  00:  IF ( _execute_R.Q )  
       THEN
         // Check function is supported and parameter are valid ?
         IF (( CheckFunctionSupported( AxesGroup := AxesGroup )) AND
             ( CheckParameterValid   ( AxesGroup := AxesGroup )))      
         THEN
           // set busy flag
           Busy := TRUE;
           // Reset command outputs
           SysDepMemSet(pDest := ADR(OutCmd), Value := 0, DataLen := SIZEOF(OutCmd));         
           // apply command parameter
          _parCmd := ParCmd;
           // init parameter sequence
          _command.ParSeq := 1;
           // create command data
           CommandData := CreateCommandPayload(AxesGroup := AxesGroup);
           // Add command to active command register
          _uniqueID := AxesGroup.Acyclic.ActiveCommandRegister.AddCmd( pCommandFB := ADR(THIS^ ));     
           // set timeout
           SetTimeout(PT := _timeoutCmd, rTimer := _timerCmd);
           // inc step counter
          _stepCmd := _stepCmd + 1;
         END_IF 
       END_IF
     

  01:  // Wait for responce received
       IF ( _responseReceived )
       THEN
         // reset response received flag
        _responseReceived := FALSE;

         CASE  _response.State 
         OF
           CmdMessageState.BUFFERED : CommandBuffered := TRUE;
           CmdMessageState.DONE     : Done            := TRUE;
           CmdMessageState.ERROR    : Error           := TRUE;
         END_CASE
                
         // Done, Aborted or Error ?
         IF (_response.State >= CmdMessageState.DONE )
         THEN
           // Reset Busy flag
           Busy := FALSE;
           // Update results
           OutCmd.TransformedPosition := _response.TransformedPosition;
           // set timeout
           SetTimeout(PT := _timeoutCmd, rTimer := _timerCmd);
           // inc step counter
          _stepCmd := _stepCmd + 1; 
         END_IF
       END_IF


  02: IF ( NOT Execute)
      THEN
        Reset();  
      END_IF     
ELSE
  // invalid step
  ErrorID := RobotLibraryEvents.ERR_INVALID_STEP;
END_CASE



// Reset FB
IF ( NOT Execute )
THEN
  Reset();  
END_IF
END_METHOD

METHOD INTERNAL ParseResponsePayload : DINT
VAR_INPUT
  /// Response data
  ResponseData : RobotLibraryRecvDataFB;
  /// Timestamp
  Timestamp    : SystemTime;  
END_VAR
// Table 6-669: Received CMD payload (RC to PLC) of "ShiftPosition"
// --------------------------
// Header
// --------------------------
// Byte 00 : USINT - ParSeq | State     
// Byte 01 : SINT  - AlarmMessageSeverity    
// Byte 02 : UINT  - AlarmMessageCode HB
// Byte 03 :       - AlarmMessageCode LB
// --------------------------
// Datablock
// --------------------------
// Byte 04  : REAL      - TransformedPosition.X HW HB
// Byte 05  :           - TransformedPosition.X HW LB
// Byte 06  :           - TransformedPosition.X LW HB
// Byte 07  :           - TransformedPosition.X LW LB
// Byte 08  : REAL      - TransformedPosition.Y HW HB
// Byte 09  :           - TransformedPosition.Y HW LB
// Byte 10  :           - TransformedPosition.Y LW HB
// Byte 11  :           - TransformedPosition.Y LW LB
// Byte 12  : REAL      - TransformedPosition.Z HW HB
// Byte 13  :           - TransformedPosition.Z HW LB
// Byte 14  :           - TransformedPosition.Z LW HB
// Byte 15  :           - TransformedPosition.Z LW LB
// Byte 16  : REAL      - TransformedPosition.RX HW HB
// Byte 17  :           - TransformedPosition.RX HW LB
// Byte 18  :           - TransformedPosition.RX LW HB
// Byte 19  :           - TransformedPosition.RX LW LB
// Byte 20  : REAL      - TransformedPosition.RY HW HB
// Byte 21  :           - TransformedPosition.RY HW LB
// Byte 22  :           - TransformedPosition.RY LW HB
// Byte 23  :           - TransformedPosition.RY LW LB
// Byte 24  : REAL      - TransformedPosition.RZ HW HB
// Byte 25  :           - TransformedPosition.RZ HW LB
// Byte 26  :           - TransformedPosition.RZ LW HB
// Byte 27  :           - TransformedPosition.RZ LW LB
// Byte 28  : ArmConfig - TransformedPosition.Config
// Byte 29  :           - Reserved
// Byte 30  : TurnNumber- TransformedPosition.TurnNumber.J1 + J2  HW HB
// Byte 31  :           - TransformedPosition.TurnNumber.J3 + J4  HW LB
// Byte 32  :           - TransformedPosition.TurnNumber.J5 + J6  LW LB
// Byte 33  :           - TransformedPosition.TurnNumber.E1       LW LB
// Byte 34  : REAL      - TransformedPosition.E1 HW HB
// Byte 35  :           - TransformedPosition.E1 HW LB
// Byte 36  :           - TransformedPosition.E1 LW HB
// Byte 37  :           - TransformedPosition.E1 LW LB
// Byte 38  : REAL      - TransformedPosition.E2 HW HB
// Byte 39  :           - TransformedPosition.E2 HW LB
// Byte 40  :           - TransformedPosition.E2 LW HB
// Byte 41  :           - TransformedPosition.E2 LW LB
// Byte 42  : REAL      - TransformedPosition.E3 HW HB
// Byte 43  :           - TransformedPosition.E3 HW LB
// Byte 44  :           - TransformedPosition.E3 LW HB
// Byte 45  :           - TransformedPosition.E3 LW LB
// Byte 46  : REAL      - TransformedPosition.E4 HW HB
// Byte 47  :           - TransformedPosition.E4 HW LB
// Byte 48  :           - TransformedPosition.E4 LW HB
// Byte 49  :           - TransformedPosition.E4 LW LB
// Byte 50  : REAL      - TransformedPosition.E5 HW HB
// Byte 51  :           - TransformedPosition.E5 HW LB
// Byte 52  :           - TransformedPosition.E5 LW HB
// Byte 53  :           - TransformedPosition.E5 LW LB
// Byte 54  : REAL      - TransformedPosition.E6 HW HB
// Byte 55  :           - TransformedPosition.E6 HW LB
// Byte 56  :           - TransformedPosition.E6 LW HB
// Byte 57  :           - TransformedPosition.E6 LW LB
// call base implementation to parse the header from payload buffer
ResponseData.PayloadPtr := SUPER^.ParseResponsePayload(ResponseData := ResponseData, Timestamp := Timestamp);

// copy parsed header to response
_response.ParSeq               := _rspHeader.ParSeq;
_response.State                := _rspHeader.State;
_response.AlarmMessageSeverity := _rspHeader.AlarmMessageSeverity;
_response.AlarmMessageCode     := _rspHeader.AlarmMessageCode;

// Get Response.TransformedPosition.X
_response.TransformedPosition.X := ResponseData.GetReal();
// Get Response.TransformedPosition.Y
_response.TransformedPosition.Y := ResponseData.GetReal();
// Get Response.TransformedPosition.Z
_response.TransformedPosition.Z := ResponseData.GetReal();
// Get Response.TransformedPosition.Rx
_response.TransformedPosition.Rx := ResponseData.GetReal();
// Get Response.TransformedPosition.Ry
_response.TransformedPosition.Ry := ResponseData.GetReal();
// Get Response.TransformedPosition.Rz
_response.TransformedPosition.Rz := ResponseData.GetReal();
// Get Response.TransformedPosition.Config
_response.TransformedPosition.Config := ResponseData.GetArmConfig();
// Get Response.TransformedPosition.TurnNumber
_response.TransformedPosition.TurnNumber := ResponseData.GetTurnNumbers();
// Get Response.TransformedPosition.E1
_response.TransformedPosition.E1 := ResponseData.GetReal();
// Get Response.TransformedPosition.E2
_response.TransformedPosition.E2 := ResponseData.GetReal();
// Get Response.TransformedPosition.E3
_response.TransformedPosition.E3 := ResponseData.GetReal();
// Get Response.TransformedPosition.E4
_response.TransformedPosition.E4 := ResponseData.GetReal();
// Get Response.TransformedPosition.E5
_response.TransformedPosition.E5 := ResponseData.GetReal();
// Get Response.TransformedPosition.E6
_response.TransformedPosition.E6 := ResponseData.GetReal();

// Create logging
ParseResponsePayloadLog(ResponseData := ResponseData, Timestamp := Timestamp);
END_METHOD

METHOD INTERNAL ParseResponsePayloadLog
VAR_INPUT
  /// Response data
  ResponseData : RobotLibraryRecvDataFB;
  /// Timestamp
  Timestamp    : SystemTime;  
END_VAR
// Create log entry for Parameter start
CreateLogMessage      ( Timestamp   := Timestamp,
                        MessageType := MessageType.CMD,
                        Severity    := Severity.DEBUG,
                        MessageCode := 0,
                        MessageText := 'Parsed the following parameter(s) from response data:');
                        
// Create log entry for TransformedPosition.X
CreateLogMessagePara1 ( Timestamp   := Timestamp,
                        MessageType := MessageType.CMD,
                        Severity    := Severity.DEBUG,
                        MessageCode := 0,
                        MessageText := 'Response.TransformedPosition.X = {1}',
                        Para1       :=  REAL_TO_STRING(_response.TransformedPosition.X));

// Create log entry for TransformedPosition.Y
CreateLogMessagePara1 ( Timestamp   := Timestamp,
                        MessageType := MessageType.CMD,
                        Severity    := Severity.DEBUG,
                        MessageCode := 0,
                        MessageText := 'Response.TransformedPosition.Y = {1}',
                        Para1       :=  REAL_TO_STRING(_response.TransformedPosition.Y));

// Create log entry for TransformedPosition.Z
CreateLogMessagePara1 ( Timestamp   := Timestamp,
                        MessageType := MessageType.CMD,
                        Severity    := Severity.DEBUG,
                        MessageCode := 0,
                        MessageText := 'Response.TransformedPosition.Z = {1}',
                        Para1       :=  REAL_TO_STRING(_response.TransformedPosition.Z));

// Create log entry for TransformedPosition.Rx
CreateLogMessagePara1 ( Timestamp   := Timestamp,
                        MessageType := MessageType.CMD,
                        Severity    := Severity.DEBUG,
                        MessageCode := 0,
                        MessageText := 'Response.TransformedPosition.Rx = {1}',
                        Para1       :=  REAL_TO_STRING(_response.TransformedPosition.Rx));

// Create log entry for TransformedPosition.Ry
CreateLogMessagePara1 ( Timestamp   := Timestamp,
                        MessageType := MessageType.CMD,
                        Severity    := Severity.DEBUG,
                        MessageCode := 0,
                        MessageText := 'Response.TransformedPosition.Ry = {1}',
                        Para1       :=  REAL_TO_STRING(_response.TransformedPosition.Ry));

// Create log entry for TransformedPosition.Rz
CreateLogMessagePara1 ( Timestamp   := Timestamp,
                        MessageType := MessageType.CMD,
                        Severity    := Severity.DEBUG,
                        MessageCode := 0,
                        MessageText := 'Response.TransformedPosition.Rz = {1}',
                        Para1       :=  REAL_TO_STRING(_response.TransformedPosition.Rz));


// Create log entry for TransformedPosition.Config
CreateLogMessagePara1 ( Timestamp   := Timestamp,
                        MessageType := MessageType.CMD,
                        Severity    := Severity.DEBUG,
                        MessageCode := 0,
                        MessageText := 'Response.TransformedPosition.Config = {1}',
                        Para1       :=  ARM_CONFIG_TO_STRING(_response.TransformedPosition.Config));

// Create log entry for TransformedPosition.TurnNumber.J1Turns
CreateLogMessagePara1 ( Timestamp   := Timestamp,
                        MessageType := MessageType.CMD,
                        Severity    := Severity.DEBUG,
                        MessageCode := 0,
                        MessageText := 'Response.TransformedPosition.TurnNumber.J1Turns = {1}',
                        Para1       :=  SINT_TO_STRING(_response.TransformedPosition.TurnNumber.J1Turns));

// Create log entry for TransformedPosition.TurnNumber.J2Turns
CreateLogMessagePara1 ( Timestamp   := Timestamp,
                        MessageType := MessageType.CMD,
                        Severity    := Severity.DEBUG,
                        MessageCode := 0,
                        MessageText := 'Response.TransformedPosition.TurnNumber.J2Turns = {1}',
                        Para1       :=  SINT_TO_STRING(_response.TransformedPosition.TurnNumber.J2Turns));

// Create log entry for TransformedPosition.TurnNumber.J3Turns
CreateLogMessagePara1 ( Timestamp   := Timestamp,
                        MessageType := MessageType.CMD,
                        Severity    := Severity.DEBUG,
                        MessageCode := 0,
                        MessageText := 'Response.TransformedPosition.TurnNumber.J3Turns = {1}',
                        Para1       :=  SINT_TO_STRING(_response.TransformedPosition.TurnNumber.J3Turns));

// Create log entry for TransformedPosition.TurnNumber.J4Turns
CreateLogMessagePara1 ( Timestamp   := Timestamp,
                        MessageType := MessageType.CMD,
                        Severity    := Severity.DEBUG,
                        MessageCode := 0,
                        MessageText := 'Response.TransformedPosition.TurnNumber.J4Turns = {1}',
                        Para1       :=  SINT_TO_STRING(_response.TransformedPosition.TurnNumber.J4Turns));

// Create log entry for TransformedPosition.TurnNumber.J5Turns
CreateLogMessagePara1 ( Timestamp   := Timestamp,
                        MessageType := MessageType.CMD,
                        Severity    := Severity.DEBUG,
                        MessageCode := 0,
                        MessageText := 'Response.TransformedPosition.TurnNumber.J5Turns = {1}',
                        Para1       :=  SINT_TO_STRING(_response.TransformedPosition.TurnNumber.J5Turns));

// Create log entry for TransformedPosition.TurnNumber.J6Turns
CreateLogMessagePara1 ( Timestamp   := Timestamp,
                        MessageType := MessageType.CMD,
                        Severity    := Severity.DEBUG,
                        MessageCode := 0,
                        MessageText := 'Response.TransformedPosition.TurnNumber.J6Turns = {1}',
                        Para1       :=  SINT_TO_STRING(_response.TransformedPosition.TurnNumber.J6Turns));

// Create log entry for TransformedPosition.TurnNumber.E1Turns
CreateLogMessagePara1 ( Timestamp   := Timestamp,
                        MessageType := MessageType.CMD,
                        Severity    := Severity.DEBUG,
                        MessageCode := 0,
                        MessageText := 'Response.TransformedPosition.TurnNumber.E1Turns = {1}',
                        Para1       :=  SINT_TO_STRING(_response.TransformedPosition.TurnNumber.E1Turns));

// Create log entry for TransformedPosition.E1
CreateLogMessagePara1 ( Timestamp   := Timestamp,
                        MessageType := MessageType.CMD,
                        Severity    := Severity.DEBUG,
                        MessageCode := 0,
                        MessageText := 'Response.TransformedPosition.E1 = {1}',
                        Para1       :=  REAL_TO_STRING(_response.TransformedPosition.E1));

// Create log entry for TransformedPosition.E2
CreateLogMessagePara1 ( Timestamp   := Timestamp,
                        MessageType := MessageType.CMD,
                        Severity    := Severity.DEBUG,
                        MessageCode := 0,
                        MessageText := 'Response.TransformedPosition.E2 = {1}',
                        Para1       :=  REAL_TO_STRING(_response.TransformedPosition.E2));

// Create log entry for TransformedPosition.E3
CreateLogMessagePara1 ( Timestamp   := Timestamp,
                        MessageType := MessageType.CMD,
                        Severity    := Severity.DEBUG,
                        MessageCode := 0,
                        MessageText := 'Response.TransformedPosition.E3 = {1}',
                        Para1       :=  REAL_TO_STRING(_response.TransformedPosition.E3));

// Create log entry for TransformedPosition.E4
CreateLogMessagePara1 ( Timestamp   := Timestamp,
                        MessageType := MessageType.CMD,
                        Severity    := Severity.DEBUG,
                        MessageCode := 0,
                        MessageText := 'Response.TransformedPosition.E4 = {1}',
                        Para1       :=  REAL_TO_STRING(_response.TransformedPosition.E4));

// Create log entry for TransformedPosition.E5
CreateLogMessagePara1 ( Timestamp   := Timestamp,
                        MessageType := MessageType.CMD,
                        Severity    := Severity.DEBUG,
                        MessageCode := 0,
                        MessageText := 'Response.TransformedPosition.E5 = {1}',
                        Para1       :=  REAL_TO_STRING(_response.TransformedPosition.E5));

// Create log entry for TransformedPosition.E6
CreateLogMessagePara1 ( Timestamp   := Timestamp,
                        MessageType := MessageType.CMD,
                        Severity    := Severity.DEBUG,
                        MessageCode := 0,
                        MessageText := 'Response.TransformedPosition.E6 = {1}',
                        Para1       :=  REAL_TO_STRING(_response.TransformedPosition.E6));
END_METHOD

METHOD PROTECTED Reset : DINT
VAR_INPUT
END_VAR
Reset := SUPER^.Reset();

Done               := FALSE;
Busy               := FALSE;
CommandBuffered    := FALSE;
END_METHOD

END_FUNCTION_BLOCK

// Library/POUs/Additional/MC_SoftSwitchTcp/MC_SoftSwitchTcpFB
/// Push robot: Robot calculates opposite vector and moves slowly in that direction
FUNCTION_BLOCK MC_SoftSwitchTcpFB EXTENDS RobotLibraryBaseExecuteFB
// ------------------------------------------------------------------------- 
//  SRCI Robot Library                                                
// ------------------------------------------------------------------------- 
//                                                                           
//  Object:      SoftSwitchTcpFB                                       
//  Author:      Thorsten Brach                                                
//  Date:        2024-06-01
//
//  Description:                                              
//   
//                                                                           
//  Copyright: 
//    (C) 2024 Thorsten Brach. All rights reserved                                                                                                                                            
//             Licensed under the LGPL-3.0 license.
//                                                                           
//  Disclaimer:                                                                           
//    This project is provided without any guarantee and can be used for   
//    private and commercial purposes. Any use is at the user’s 
//    own risk and responsibility.
//
// -------------------------------------------------------------------------
VAR_INPUT
  /// Parameter which determines the behavior towards the previously sent and still active or buffered commands
  AbortingMode       : AbortingMode;
  /// Defines the target sequence in which the command will be executed
  SequenceFlag       : SequenceFlag;   
  /// Command parameter 
  ParCmd             : SoftSwitchTcpParCmd;  
END_VAR
VAR_OUTPUT
  /// Command is transferred and confirmed by the RC
  CommandBuffered    : BOOL;
  /// The command "SoftSwitchTCP" takes control of the according axis group.
  Active             : BOOL;
  /// The command was aborted by another command
  CommandAborted     : BOOL;
  /// TRUE, while command is interrupted during execution and can be continued
  CommandInterrupted : BOOL;
  /// command results
  OutCmd             : SoftSwitchTcpOutCmd;     
END_VAR

VAR
  /// internal copy of command parameter 
 _parCmd             : SoftSwitchTcpParCmd;
  /// command data to send
 _command            : SoftSwitchTcpSendData;
  /// response data received
 _response           : SoftSwitchTcpRecvData;      
END_VAR

SUPER^(AxesGroup := AxesGroup);

METHOD PROTECTED CheckFunctionSupported : BOOL
VAR_IN_OUT
  /// Robot assignment of function
  AxesGroup : AxesGroup; 
END_VAR
CheckFunctionSupported := AxesGroup.InternalData.RCSupportedFunctions.SoftSwitchTCP;

IF ( NOT CheckFunctionSupported )
THEN
  // call base implementation for set error and create log entry
  SUPER^.CheckFunctionSupported(AxesGroup := AxesGroup);
END_IF
END_METHOD

METHOD PROTECTED CheckParameterChanged : BOOL
VAR_IN_OUT
  /// Robot assignment of function
  AxesGroup    : AxesGroup; 
END_VAR
// Check ParCmd Size is > 0, because MemCmp does not work correctly with size = 0
IF (SIZEOF(ParCmd) = 0) 
THEN 
  RETURN;
END_IF

// compare memory 
_parameterChanged := ( SysDepMemCmp(pData1 := ADR(ParCmd), pData2 := ADR(_parCmd), DataLen := SIZEOF(ParCmd)) <> RobotLibraryConstants.OK );

// check parameter valid ?
_parameterValid   := CheckParameterValid( AxesGroup := AxesGroup );

IF ((  _parameterChanged        )  AND 
    (  _parameterValid          )) OR
    (  _parameterUpdateInternal )  
THEN  
  // reset internal flag for send parameter update
 _parameterUpdateInternal := FALSE;
  // update internal copy of parameters 
 _parCmd := ParCmd;
  // inc parameter sequence
 _command.ParSeq := _command.ParSeq + 1;
  // update command data  
  CommandData := CreateCommandPayload(AxesGroup := AxesGroup); // ( Access via reference to rCommandFB in ACR )
  // notify active command register 
  AxesGroup.Acyclic.ActiveCommandRegister.NotifyParameterChanged := _uniqueID;
END_IF
END_METHOD

METHOD INTERNAL CreateCommandPayload : RobotLibrarySendDataFB
VAR_IN_OUT
  /// Robot assignment of function
  AxesGroup : AxesGroup; 
END_VAR
// Table 6-748: Sent CMD payload (PLC to RC) of "SoftSwitchTCP"
// --------------------------
// Header
// --------------------------
// Byte 00 : UINT  - Type HB     
// Byte 01 :       - Type LB    
// Byte 02 : USINT - Reserve | ExecutionMode
// Byte 03 : USINT - ParSeq  | Priority
// --------------------------
// Datablock
// --------------------------
// Byte 04 : USINT  - LimitMode
// Byte 05 : BYTE   - CompliantAxes
// Byte 06 : BOOL   - ReferenceType
// Byte 07 : USINT  - ReferenceNo
// Byte 08 : INT    - ResistanceForceTCP HW HB
// Byte 09 :        - ResistanceForceTCP HW LB
// Byte 10 : UINT   - ResistanceForceAxis[0] HW HB
// Byte 11 :        - ResistanceForceAxis[0] HW LB
// Byte 12 : UINT   - ResistanceForceAxis[1] HW HB
// Byte 13 :        - ResistanceForceAxis[1] HW LB
// Byte 14 : UINT   - ResistanceForceAxis[2] HW HB
// Byte 15 :        - ResistanceForceAxis[2] HW LB
// Byte 16 : UINT   - ResistanceForceAxis[3] HW HB
// Byte 17 :        - ResistanceForceAxis[3] HW LB
// Byte 18 : UINT   - ResistanceForceAxis[4] HW HB
// Byte 19 :        - ResistanceForceAxis[4] HW LB
// Byte 20 : UINT   - ResistanceForceAxis[5] HW HB
// Byte 21 :        - ResistanceForceAxis[5] HW LB
// Byte 22 : REAL   - VectorData[0] HW HB
// Byte 23 :        - VectorData[0] HW LB
// Byte 24 :        - VectorData[0] LW HB
// Byte 25 :        - VectorData[0] LW LB
// Byte 26 : REAL   - VectorData[1] HW HB
// Byte 27 :        - VectorData[1] HW LB
// Byte 28 :        - VectorData[1] LW HB
// Byte 29 :        - VectorData[1] LW LB
// Byte 30 : REAL   - VectorData[2] HW HB
// Byte 31 :        - VectorData[2] HW LB
// Byte 32 :        - VectorData[2] LW HB
// Byte 33 :        - VectorData[2] LW LB
// Byte 34 : REAL   - VectorData[3] HW HB
// Byte 35 :        - VectorData[3] HW LB
// Byte 36 :        - VectorData[3] LW HB
// Byte 37 :        - VectorData[3] LW LB
// Byte 38 : REAL   - VectorData[4] HW HB
// Byte 39 :        - VectorData[4] HW LB
// Byte 40 :        - VectorData[4] LW HB
// Byte 41 :        - VectorData[4] LW LB
// Byte 42 : REAL   - VectorData[5] HW HB
// Byte 43 :        - VectorData[5] HW LB
// Byte 44 :        - VectorData[5] LW HB
// Byte 45 :        - VectorData[5] LW LB
// Byte 46 : USINT  - ResistanceForceMode
// set command parameter 
_command.CmdTyp                    :=  CmdType.ShiftPosition;
_command.ExecMode                  :=  ExecMode;
_command.ParSeq                    := _command.ParSeq;
_command.Priority                  :=  Priority;

_command.LimitMode                 := _parCmd.LimitMode;
_command.CompliantAxes             := _parCmd.CompliantAxes;       
_command.ReferenceType             := _parCmd.ReferenceType;
_command.ReferenceNo               := _parCmd.ReferenceNo;
_command.ResistanceForceTCP        := REAL_TO_PERCENT_INT (_parCmd.ResistanceForceTCP     , IsOptional := TRUE );
_command.ResistanceForceMode       :=_parCmd.ResistanceForceMode;
_command.ResistanceForceAxis[0]    := REAL_TO_PERCENT_UINT(_parCmd.ResistanceForceAxis[0] , IsOptional := TRUE );
_command.ResistanceForceAxis[1]    := REAL_TO_PERCENT_UINT(_parCmd.ResistanceForceAxis[1] , IsOptional := TRUE );
_command.ResistanceForceAxis[2]    := REAL_TO_PERCENT_UINT(_parCmd.ResistanceForceAxis[2] , IsOptional := TRUE );
_command.ResistanceForceAxis[3]    := REAL_TO_PERCENT_UINT(_parCmd.ResistanceForceAxis[3] , IsOptional := TRUE );
_command.ResistanceForceAxis[4]    := REAL_TO_PERCENT_UINT(_parCmd.ResistanceForceAxis[4] , IsOptional := TRUE );
_command.ResistanceForceAxis[5]    := REAL_TO_PERCENT_UINT(_parCmd.ResistanceForceAxis[5] , IsOptional := TRUE );
_command.VectorData                :=_parCmd.VectorData;


// copy command data to header
_cmdHeader := _command;
// call base implementation to copy header to payload buffer
CreateCommandPayload := SUPER^.CreateCommandPayload(AxesGroup := AxesGroup);

// add command.LimitMode
CreateCommandPayload.AddUsint(_command.LimitMode);
// add command.CompliantAxes
CreateCommandPayload.AddByte(_command.CompliantAxes);
// add command.ReferenceType
CreateCommandPayload.AddBool(_command.ReferenceType.0);
// add command.ReferenceNo
CreateCommandPayload.AddUsint(_command.ReferenceNo);
// add command.ResistanceForceTCP
CreateCommandPayload.AddInt(_command.ResistanceForceTCP);
// add command.ResistanceForceAxis[0]
CreateCommandPayload.AddUint(_command.ResistanceForceAxis[0]);
// add command.ResistanceForceAxis[1]
CreateCommandPayload.AddUint(_command.ResistanceForceAxis[1]);
// add command.ResistanceForceAxis[2]
CreateCommandPayload.AddUint(_command.ResistanceForceAxis[2]);
// add command.ResistanceForceAxis[3]
CreateCommandPayload.AddUint(_command.ResistanceForceAxis[3]);
// add command.ResistanceForceAxis[4]
CreateCommandPayload.AddUint(_command.ResistanceForceAxis[4]);
// add command.ResistanceForceAxis[5]
CreateCommandPayload.AddUint(_command.ResistanceForceAxis[5]);
// add command.VectorData[0]
CreateCommandPayload.AddReal(_command.VectorData[0]);
// add command.VectorData[1]
CreateCommandPayload.AddReal(_command.VectorData[1]);
// add command.VectorData[2]
CreateCommandPayload.AddReal(_command.VectorData[2]);
// add command.VectorData[3]
CreateCommandPayload.AddReal(_command.VectorData[3]);
// add command.VectorData[4]
CreateCommandPayload.AddReal(_command.VectorData[4]);
// add command.VectorData[5]
CreateCommandPayload.AddReal(_command.VectorData[5]);
// add command.ResistanceForceMode
CreateCommandPayload.AddUsint(_command.ResistanceForceMode);

// Create logging
CreateCommandPayloadLog(AxesGroup := AxesGroup);
END_METHOD

METHOD INTERNAL CreateCommandPayloadLog
VAR_IN_OUT
  /// Robot assignment of function
  AxesGroup : AxesGroup; 
END_VAR
// Create log entry for Parameter start
CreateLogMessage      ( Timestamp   := AxesGroup.InternalData.SystemTime,
                        MessageType := MessageType.CMD,
                        Severity    := Severity.DEBUG,
                        MessageCode := 0,
                        MessageText := 'Create command payload with the following parameter(s) :');
  
// Create log entry for LimitMode
CreateLogMessagePara1 ( Timestamp   := AxesGroup.InternalData.SystemTime,
                        MessageType := MessageType.CMD,
                        Severity    := Severity.DEBUG,
                        MessageCode := 0,
                        MessageText := 'Command.LimitMode = {1}',
                        Para1       :=  LIMIT_MODE_TO_STRING(_command.LimitMode));

// Create log entry for CompliantAxes
CreateLogMessagePara1 ( Timestamp   := AxesGroup.InternalData.SystemTime,
                        MessageType := MessageType.CMD,
                        Severity    := Severity.DEBUG,
                        MessageCode := 0,
                        MessageText := 'Command.CompliantAxes = {1}',
                        Para1       :=  BYTE_TO_STRING(_command.CompliantAxes));

// Create log entry for ReferenceType
CreateLogMessagePara1 ( Timestamp   := AxesGroup.InternalData.SystemTime,
                        MessageType := MessageType.CMD,
                        Severity    := Severity.DEBUG,
                        MessageCode := 0,
                        MessageText := 'Command.ReferenceType = {1}',
                        Para1       :=  BYTE_TO_STRING_BIN(_command.ReferenceType));

// Create log entry for ReferenceNo
CreateLogMessagePara1 ( Timestamp   := AxesGroup.InternalData.SystemTime,
                        MessageType := MessageType.CMD,
                        Severity    := Severity.DEBUG,
                        MessageCode := 0,
                        MessageText := 'Command.ReferenceNo = {1}',
                        Para1       :=  USINT_TO_STRING(_command.ReferenceNo));

// Create log entry for ResistanceForceTCP
CreateLogMessagePara1 ( Timestamp   := AxesGroup.InternalData.SystemTime,
                        MessageType := MessageType.CMD,
                        Severity    := Severity.DEBUG,
                        MessageCode := 0,
                        MessageText := 'Command.ResistanceForceTCP = {1}',
                        Para1       :=  INT_TO_STRING(_command.ResistanceForceTCP));

// Create log entry for ResistanceForceAxis[0]
CreateLogMessagePara1 ( Timestamp   := AxesGroup.InternalData.SystemTime,
                        MessageType := MessageType.CMD,
                        Severity    := Severity.DEBUG,
                        MessageCode := 0,
                        MessageText := 'Command.ResistanceForceAxis[0] = {1}',
                        Para1       :=  UINT_TO_STRING(_command.ResistanceForceAxis[0]));

// Create log entry for ResistanceForceAxis[1]
CreateLogMessagePara1 ( Timestamp   := AxesGroup.InternalData.SystemTime,
                        MessageType := MessageType.CMD,
                        Severity    := Severity.DEBUG,
                        MessageCode := 0,
                        MessageText := 'Command.ResistanceForceAxis[1] = {1}',
                        Para1       :=  UINT_TO_STRING(_command.ResistanceForceAxis[1]));

// Create log entry for ResistanceForceAxis[2]
CreateLogMessagePara1 ( Timestamp   := AxesGroup.InternalData.SystemTime,
                        MessageType := MessageType.CMD,
                        Severity    := Severity.DEBUG,
                        MessageCode := 0,
                        MessageText := 'Command.ResistanceForceAxis[2] = {1}',
                        Para1       :=  UINT_TO_STRING(_command.ResistanceForceAxis[2]));

// Create log entry for ResistanceForceAxis[3]
CreateLogMessagePara1 ( Timestamp   := AxesGroup.InternalData.SystemTime,
                        MessageType := MessageType.CMD,
                        Severity    := Severity.DEBUG,
                        MessageCode := 0,
                        MessageText := 'Command.ResistanceForceAxis[3] = {1}',
                        Para1       :=  UINT_TO_STRING(_command.ResistanceForceAxis[3]));

// Create log entry for ResistanceForceAxis[4]
CreateLogMessagePara1 ( Timestamp   := AxesGroup.InternalData.SystemTime,
                        MessageType := MessageType.CMD,
                        Severity    := Severity.DEBUG,
                        MessageCode := 0,
                        MessageText := 'Command.ResistanceForceAxis[4] = {1}',
                        Para1       :=  UINT_TO_STRING(_command.ResistanceForceAxis[4]));

// Create log entry for ResistanceForceAxis[5]
CreateLogMessagePara1 ( Timestamp   := AxesGroup.InternalData.SystemTime,
                        MessageType := MessageType.CMD,
                        Severity    := Severity.DEBUG,
                        MessageCode := 0,
                        MessageText := 'Command.ResistanceForceAxis[5] = {1}',
                        Para1       :=  UINT_TO_STRING(_command.ResistanceForceAxis[5]));

// Create log entry for VectorData[0]
CreateLogMessagePara1 ( Timestamp   := AxesGroup.InternalData.SystemTime,
                        MessageType := MessageType.CMD,
                        Severity    := Severity.DEBUG,
                        MessageCode := 0,
                        MessageText := 'Command.VectorData[0] = {1}',
                        Para1       :=  REAL_TO_STRING(_command.VectorData[0]));
                        
// Create log entry for VectorData[1]
CreateLogMessagePara1 ( Timestamp   := AxesGroup.InternalData.SystemTime,
                        MessageType := MessageType.CMD,
                        Severity    := Severity.DEBUG,
                        MessageCode := 0,
                        MessageText := 'Command.VectorData[1] = {1}',
                        Para1       :=  REAL_TO_STRING(_command.VectorData[1]));

// Create log entry for VectorData[2]
CreateLogMessagePara1 ( Timestamp   := AxesGroup.InternalData.SystemTime,
                        MessageType := MessageType.CMD,
                        Severity    := Severity.DEBUG,
                        MessageCode := 0,
                        MessageText := 'Command.VectorData[2] = {1}',
                        Para1       :=  REAL_TO_STRING(_command.VectorData[2]));

// Create log entry for VectorData[3]
CreateLogMessagePara1 ( Timestamp   := AxesGroup.InternalData.SystemTime,
                        MessageType := MessageType.CMD,
                        Severity    := Severity.DEBUG,
                        MessageCode := 0,
                        MessageText := 'Command.VectorData[3] = {1}',
                        Para1       :=  REAL_TO_STRING(_command.VectorData[3]));

// Create log entry for VectorData[4]
CreateLogMessagePara1 ( Timestamp   := AxesGroup.InternalData.SystemTime,
                        MessageType := MessageType.CMD,
                        Severity    := Severity.DEBUG,
                        MessageCode := 0,
                        MessageText := 'Command.VectorData[4] = {1}',
                        Para1       :=  REAL_TO_STRING(_command.VectorData[4]));

// Create log entry for VectorData[5]
CreateLogMessagePara1 ( Timestamp   := AxesGroup.InternalData.SystemTime,
                        MessageType := MessageType.CMD,
                        Severity    := Severity.DEBUG,
                        MessageCode := 0,
                        MessageText := 'Command.VectorData[5] = {1}',
                        Para1       :=  REAL_TO_STRING(_command.VectorData[5]));
                        
// Create log entry for ResistanceForceMode
CreateLogMessagePara1 ( Timestamp   := AxesGroup.InternalData.SystemTime,
                        MessageType := MessageType.CMD,
                        Severity    := Severity.DEBUG,
                        MessageCode := 0,
                        MessageText := 'Command.ResistanceForceMode = {1}',
                        Para1       :=  USINT_TO_STRING(_command.ResistanceForceMode));
END_METHOD

METHOD FB_init : BOOL
VAR_INPUT
  /// if TRUE, the retain variables are initialized (warm start / cold start)
  bInitRetains : BOOL; 
  /// if TRUE, the instance afterwards gets moved into the copy code (online change)
  bInCopyCode  : BOOL;  
END_VAR
MyType := 'MC_SoftSwitchTcpFB';
END_METHOD

METHOD PROTECTED OnCall
VAR_IN_OUT
  /// Robot assignment of function
  AxesGroup : AxesGroup; 
END_VAR
// call base implementation
SUPER^.OnCall(AxesGroup := AxesGroup);

CASE _stepCmd OF
  
  00:  IF ( _execute_R.Q )  
       THEN
         // Check function is supported and parameter are valid ?
         IF (( CheckFunctionSupported( AxesGroup := AxesGroup )) AND
             ( CheckParameterValid   ( AxesGroup := AxesGroup )))      
         THEN
           // set busy flag
           Busy := TRUE;
           // Reset command outputs
           SysDepMemSet(pDest := ADR(OutCmd), Value := 0, DataLen := SIZEOF(OutCmd));         
           // apply command parameter
          _parCmd := ParCmd;
           // init parameter sequence
          _command.ParSeq := 1;
           // create command data
           CommandData := CreateCommandPayload(AxesGroup := AxesGroup);
           // Add command to active command register
          _uniqueID := AxesGroup.Acyclic.ActiveCommandRegister.AddCmd( pCommandFB := ADR(THIS^ ));     
           // set timeout
           SetTimeout(PT := _timeoutCmd, rTimer := _timerCmd);
           // inc step counter
          _stepCmd := _stepCmd + 1;
         END_IF 
       END_IF
     

  01:  // Wait for responce received
       IF ( _responseReceived )
       THEN
         // reset response received flag
        _responseReceived := FALSE;
         // reset Active flag
         Active := FALSE;
         
         CASE  _response.State 
         OF
           CmdMessageState.BUFFERED    : CommandBuffered    := TRUE;
           CmdMessageState.ACTIVE      : Active             := TRUE;           
           CmdMessageState.INTERRUPTED : CommandInterrupted := TRUE;
           CmdMessageState.DONE        : Done               := TRUE;           
           CmdMessageState.ABORTED     : CommandAborted     := TRUE;
           CmdMessageState.ERROR       : Error              := TRUE;
         END_CASE
                
         // Done, Aborted or Error ?
         IF (_response.State >= CmdMessageState.DONE )
         THEN
           // Reset Busy flag
           Busy := FALSE;
           // Update results
           OutCmd.SoftMovement := _response.SoftMovement;
           // set timeout
           SetTimeout(PT := _timeoutCmd, rTimer := _timerCmd);
           // inc step counter
          _stepCmd := _stepCmd + 1; 
         END_IF
       END_IF


  02: IF ( NOT Execute)
      THEN
        Reset();
      END_IF     
ELSE
  // invalid step
  ErrorID := RobotLibraryEvents.ERR_INVALID_STEP;
END_CASE


// Reset FB
IF ( NOT Execute )
THEN
  Reset();  
END_IF
END_METHOD

METHOD INTERNAL ParseResponsePayload : DINT
VAR_INPUT
  /// Response data
  ResponseData : RobotLibraryRecvDataFB;
  /// Timestamp
  Timestamp    : SystemTime;  
END_VAR
// Table 6-749: Received CMD payload (RC to PLC) of "SoftSwitchTCP"
// --------------------------
// Header
// --------------------------
// Byte 00 : USINT - ParSeq | State     
// Byte 01 : SINT  - AlarmMessageSeverity    
// Byte 02 : UINT  - AlarmMessageCode HB
// Byte 03 :       - AlarmMessageCode LB
// --------------------------
// Datablock
// --------------------------
// Byte 04  : BOOL - SoftMovement
// call base implementation to parse the header from payload buffer
ResponseData.PayloadPtr := SUPER^.ParseResponsePayload(ResponseData := ResponseData, Timestamp := Timestamp);

// copy parsed header to response
_response.ParSeq               := _rspHeader.ParSeq;
_response.State                := _rspHeader.State;
_response.AlarmMessageSeverity := _rspHeader.AlarmMessageSeverity;
_response.AlarmMessageCode     := _rspHeader.AlarmMessageCode;

// Get Response.SoftMovement
_response.SoftMovement := ResponseData.GetBool();

// Create logging
ParseResponsePayloadLog(ResponseData := ResponseData, Timestamp := Timestamp);
END_METHOD

METHOD INTERNAL ParseResponsePayloadLog
VAR_INPUT
  /// Response data
  ResponseData : RobotLibraryRecvDataFB;
  /// Timestamp
  Timestamp    : SystemTime;  
END_VAR
// Create log entry for Parameter start
CreateLogMessage      ( Timestamp   := Timestamp,
                        MessageType := MessageType.CMD,
                        Severity    := Severity.DEBUG,
                        MessageCode := 0,
                        MessageText := 'Parsed the following parameter(s) from response data:');
                        
// Create log entry for SoftMovement
CreateLogMessagePara1 ( Timestamp   := Timestamp,
                        MessageType := MessageType.CMD,
                        Severity    := Severity.DEBUG,
                        MessageCode := 0,
                        MessageText := 'Response.SoftMovement = {1}',
                        Para1       :=  BOOL_TO_STRING(_response.SoftMovement));
END_METHOD

METHOD PROTECTED Reset : DINT
VAR_INPUT
END_VAR
Reset := SUPER^.Reset();

Done               := FALSE;
Busy               := FALSE;
Active             := FALSE;
CommandBuffered    := FALSE;
CommandAborted     := FALSE;
CommandInterrupted := FALSE;
END_METHOD

END_FUNCTION_BLOCK

// Library/POUs/Additional/MC_StopSubprogram/MC_StopSubprogramFB
/// Stops an active subprogram
FUNCTION_BLOCK MC_StopSubprogramFB EXTENDS RobotLibraryBaseExecuteFB
// ------------------------------------------------------------------------- 
//  SRCI Robot Library                                                
// ------------------------------------------------------------------------- 
//                                                                           
//  Object:      StopSubprogramFB                                       
//  Author:      Thorsten Brach                                                
//  Date:        2024-06-01
//
//  Description:                                              
//   
//                                                                           
//  Copyright: 
//    (C) 2024 Thorsten Brach. All rights reserved                                                                                                                                            
//             Licensed under the LGPL-3.0 license.
//                                                                           
//  Disclaimer:                                                                           
//    This project is provided without any guarantee and can be used for   
//    private and commercial purposes. Any use is at the user’s 
//    own risk and responsibility.
//
// -------------------------------------------------------------------------
VAR_INPUT
  /// Defines the target sequence in which the command will be executed
  SequenceFlag      : SequenceFlag;
  /// command parameter 
  ParCmd            : StopSubprogramParCmd;
END_VAR

VAR_OUTPUT
  /// Command is transferred and confirmed by the RC
  CommandBuffered    : BOOL;
  /// The command was aborted by another command
  CommandAborted     : BOOL;
  /// TRUE, while command is interrupted during execution and can be continued.
  CommandInterrupted : BOOL;
  /// command outputs
  OutCmd             : StopSubprogramOutCmd;       
END_VAR



VAR
  /// internal copy of command parameter 
 _parCmd             : StopSubprogramParCmd;
  /// command data to send
 _command            : StopSubprogramSendData;
  /// response data received
 _response           : StopSubprogramRecvData;      
END_VAR

SUPER^(AxesGroup := AxesGroup);

METHOD PROTECTED CheckFunctionSupported : BOOL
VAR_IN_OUT
  /// Robot assignment of function
  AxesGroup : AxesGroup; 
END_VAR
CheckFunctionSupported := AxesGroup.InternalData.RCSupportedFunctions.StopSubprogram;

IF ( NOT CheckFunctionSupported )
THEN
  // call base implementation for set error and create log entry
  SUPER^.CheckFunctionSupported(AxesGroup := AxesGroup);
END_IF
END_METHOD

METHOD PROTECTED CheckParameterChanged : BOOL
VAR_IN_OUT
  /// Robot assignment of function
  AxesGroup    : AxesGroup; 
END_VAR
// Check ParCmd Size is > 0, because MemCmp does not work correctly with size = 0
IF (SIZEOF(ParCmd) = 0) 
THEN 
  RETURN;
END_IF

// compare memory 
_parameterChanged := ( SysDepMemCmp(pData1 := ADR(ParCmd), pData2 := ADR(_parCmd), DataLen := SIZEOF(ParCmd)) <> RobotLibraryConstants.OK );

// check parameter valid ?
_parameterValid   := CheckParameterValid( AxesGroup := AxesGroup );

IF ((  _parameterChanged        )  AND 
    (  _parameterValid          )) OR
    (  _parameterUpdateInternal )  
THEN  
  // reset internal flag for send parameter update
 _parameterUpdateInternal := FALSE;
  // update internal copy of parameters 
 _parCmd := ParCmd;
  // inc parameter sequence
 _command.ParSeq := _command.ParSeq + 1;
  // update command data  
  CommandData := CreateCommandPayload(AxesGroup := AxesGroup); // ( Access via reference to rCommandFB in ACR )
  // notify active command register 
  AxesGroup.Acyclic.ActiveCommandRegister.NotifyParameterChanged := _uniqueID;
END_IF
END_METHOD

METHOD INTERNAL CreateCommandPayload : RobotLibrarySendDataFB
VAR_IN_OUT
  /// Robot assignment of function
  AxesGroup : AxesGroup; 
END_VAR
// Table 6-697: Sent CMD payload (PLC to RC) of "StopSubprogram"
// --------------------------
// Header
// --------------------------
// Byte 00 : UINT  - Type HB     
// Byte 01 :       - Type LB    
// Byte 02 : USINT - Reserve | ExecutionMode
// Byte 03 : USINT - ParSeq  | Priority
// --------------------------
// Datablock
// --------------------------
// Byte 04 : SINT  EmitterID[0];
// Byte 05 : SINT  EmitterID[1];
// Byte 06 : SINT  EmitterID[2];
// Byte 07 : SINT  EmitterID[3];
// Byte 08 : SINT  ListenerID;
// Byte 09 : BYTE  Reserved;
// Byte 10 : UINT  TargetID;
// Byte 11 :       TargetID;
// Byte 12 : USINT StopMode;
// set command parameter 
_command.CmdTyp     :=  CmdType.StopSubprogram;
_command.ExecMode   :=  ExecMode;
_command.ParSeq     := _command.ParSeq;
_command.Priority   :=  Priority;
_command.EmitterID  := _parCmd.EmitterID;
_command.Reserve    := 0;
_command.ListenerID := 0; {warning 'ToDo'}
_command.Reserve    := 0;
_command.TargetID   := _parCmd.TargetID;
_command.StopMode   := _parCmd.StopMode;


// copy command data to header
_cmdHeader := _command;
// call base implementation to copy header to payload buffer
CreateCommandPayload := SUPER^.CreateCommandPayload(AxesGroup := AxesGroup);

// add command.EmitterID[0]
CreateCommandPayload.AddSint(_command.EmitterID[0]);
// add command.EmitterID[1]
CreateCommandPayload.AddSint(_command.EmitterID[1]);
// add command.EmitterID[2]
CreateCommandPayload.AddSint(_command.EmitterID[2]);
// add command.EmitterID[3]
CreateCommandPayload.AddSint(_command.EmitterID[3]);
// add command.ListenerID
CreateCommandPayload.AddSint(_command.ListenerID);
// add command.Reserve
CreateCommandPayload.AddByte(_command.Reserve);
// add command.TargetID
CreateCommandPayload.AddUint(_command.TargetID);
// add command.StopMode
CreateCommandPayload.AddUsint(_command.StopMode);

// Create logging
CreateCommandPayloadLog(AxesGroup := AxesGroup);
END_METHOD

METHOD INTERNAL CreateCommandPayloadLog
VAR_IN_OUT
  /// Robot assignment of function
  AxesGroup : AxesGroup; 
END_VAR
VAR 
  /// internal index for loops
 _idx : DINT;
END_VAR
// Create log entry for Parameter start
CreateLogMessage      ( Timestamp   := AxesGroup.InternalData.SystemTime,
                        MessageType := MessageType.CMD,
                        Severity    := Severity.DEBUG,
                        MessageCode := 0,
                        MessageText := 'Create command payload with the following parameter(s) :');
  
// Create log entry for EmitterID[x]
FOR _idx := 0 TO 3
DO
  CreateLogMessagePara2 ( Timestamp   := AxesGroup.InternalData.SystemTime,
                          MessageType := MessageType.CMD,
                          Severity    := Severity.DEBUG,
                          MessageCode := 0,
                          MessageText := 'Command.EmitterID[{2}] = {1}',
                          Para1       :=  SINT_TO_STRING(_command.EmitterID[_idx]),
                          Para2       :=  DINT_TO_STRING(_idx));
END_FOR

// Create log entry for ListenerID
CreateLogMessagePara1 ( Timestamp   := AxesGroup.InternalData.SystemTime,
                        MessageType := MessageType.CMD,
                        Severity    := Severity.DEBUG,
                        MessageCode := 0,
                        MessageText := 'Command.ListenerID = {1}',
                        Para1       :=  SINT_TO_STRING(_command.ListenerID));
                        
// Create log entry for Reserve
CreateLogMessagePara1 ( Timestamp   := AxesGroup.InternalData.SystemTime,
                        MessageType := MessageType.CMD,
                        Severity    := Severity.DEBUG,
                        MessageCode := 0,
                        MessageText := 'Command.Reserve = {1}',
                        Para1       :=  BYTE_TO_STRING(_command.Reserve));
                        
// Create log entry for TargetID
CreateLogMessagePara1 ( Timestamp   := AxesGroup.InternalData.SystemTime,
                        MessageType := MessageType.CMD,
                        Severity    := Severity.DEBUG,
                        MessageCode := 0,
                        MessageText := 'Command.TargetID = {1}',
                        Para1       :=  UINT_TO_STRING(_command.TargetID));

// Create log entry for StopMode
CreateLogMessagePara1 ( Timestamp   := AxesGroup.InternalData.SystemTime,
                        MessageType := MessageType.CMD,
                        Severity    := Severity.DEBUG,
                        MessageCode := 0,
                        MessageText := 'Command.StopMode = {1}',
                        Para1       :=  STOP_MODE_TO_STRING(_command.StopMode));
END_METHOD

METHOD FB_init : BOOL
VAR_INPUT
  /// if TRUE, the retain variables are initialized (warm start / cold start)
  bInitRetains : BOOL; 
  /// if TRUE, the instance afterwards gets moved into the copy code (online change)
  bInCopyCode  : BOOL;  
END_VAR
MyType := 'MC_StopSubprogramFB';

ExecMode := ExecutionMode.PARALLEL;
END_METHOD

METHOD PROTECTED OnCall
VAR_IN_OUT
  /// Robot assignment of function
  AxesGroup : AxesGroup; 
END_VAR
// call base implementation
SUPER^.OnCall(AxesGroup := AxesGroup);

CASE _stepCmd OF
  
  00:  IF ( _execute_R.Q ) 
       THEN
         // Check function is supported and parameter are valid ?
         IF (( CheckFunctionSupported( AxesGroup := AxesGroup )) AND
             ( CheckParameterValid   ( AxesGroup := AxesGroup )))      
         THEN
           // set busy flag
           Busy := TRUE;
           // Reset command outputs
           SysDepMemSet(pDest := ADR(OutCmd), Value := 0, DataLen := SIZEOF(OutCmd));         
           // apply command parameter
          _parCmd := ParCmd;
           // init parameter sequence
          _command.ParSeq := 1;
           // create command data
           CommandData := CreateCommandPayload(AxesGroup := AxesGroup);
           // Add command to active command register
          _uniqueID := AxesGroup.Acyclic.ActiveCommandRegister.AddCmd( pCommandFB := ADR(THIS^ ));     
           // set timeout
           SetTimeout(PT := _timeoutCmd, rTimer := _timerCmd);
           // inc step counter
          _stepCmd := _stepCmd + 1;
         END_IF 
       END_IF
     

  01:  // Wait for responce received
       IF ( _responseReceived )
       THEN
         // reset response received flag
        _responseReceived := FALSE;

         CASE  _response.State 
         OF
           CmdMessageState.BUFFERED    : CommandBuffered    := TRUE;
           CmdMessageState.INTERRUPTED : CommandInterrupted := TRUE;        
           CmdMessageState.DONE        : Done               := TRUE;        
           CmdMessageState.ABORTED     : CommandAborted     := TRUE;
           CmdMessageState.ERROR       : Error              := TRUE;
         END_CASE
                
         // Done, Aborted or Error ?
         IF (_response.State >= CmdMessageState.DONE )
         THEN
           // Reset Busy flag
           Busy := FALSE;
           // Update results
           OutCmd.OriginID          := _response.OriginID;
           OutCmd.InvocationCounter := _response.InvocationCounter;
           // set timeout
           SetTimeout(PT := _timeoutCmd, rTimer := _timerCmd);
           // inc step counter
          _stepCmd := _stepCmd + 1; 
         END_IF
       END_IF


  02: IF ( NOT Execute)
      THEN
        Reset();  
      END_IF     
ELSE
  // invalid step
  ErrorID := RobotLibraryEvents.ERR_INVALID_STEP;
END_CASE


// Reset FB
IF ( NOT Execute )
THEN
  Reset();  
END_IF
END_METHOD

METHOD INTERNAL ParseResponsePayload : DINT
VAR_INPUT
  /// Response data
  ResponseData : RobotLibraryRecvDataFB;
  /// Timestamp
  Timestamp    : SystemTime;  
END_VAR
// Table 6-698: Received CMD payload (RC to PLC) of "StopSubprogram"
// --------------------------
// Header
// --------------------------
// Byte 00 : USINT   - ParSeq | State     
// Byte 01 : SINT    - AlarmMessageSeverity    
// Byte 02 : UINT    - AlarmMessageCode HB
// Byte 03 :         - AlarmMessageCode LB
// --------------------------
// Datablock
// --------------------------
// Byte 04 : USINT      - InvocationCounter
// Byte 05 : SINT       - Reserved
// Byte 06 : INT        - OriginID HW HB
// Byte 07 :            - OriginID HW LB
// call base implementation to parse the header from payload buffer
ResponseData.PayloadPtr := SUPER^.ParseResponsePayload(ResponseData := ResponseData, Timestamp := Timestamp);

// copy parsed header to response
_response.ParSeq               := _rspHeader.ParSeq;
_response.State                := _rspHeader.State;
_response.AlarmMessageSeverity := _rspHeader.AlarmMessageSeverity;
_response.AlarmMessageCode     := _rspHeader.AlarmMessageCode;

// Get Response.InvocationCounter
_response.InvocationCounter := ResponseData.GetUsint();
// Get Response.Reserve
_response.Reserve := ResponseData.GetSint();
// Get Response.OriginID
_response.OriginID := ResponseData.GetInt();

// Create logging
ParseResponsePayloadLog(ResponseData := ResponseData, Timestamp := Timestamp);
END_METHOD

METHOD INTERNAL ParseResponsePayloadLog
VAR_INPUT
  /// Response data
  ResponseData : RobotLibraryRecvDataFB;
  /// Timestamp
  Timestamp    : SystemTime;  
END_VAR
// Create log entry for Parameter start
CreateLogMessage      ( Timestamp   := Timestamp,
                        MessageType := MessageType.CMD,
                        Severity    := Severity.DEBUG,
                        MessageCode := 0,
                        MessageText := 'Parsed the following parameter(s) from response data:');
                        
// Create log entry for InvocationCounter
CreateLogMessagePara1 ( Timestamp   := Timestamp,
                        MessageType := MessageType.CMD,
                        Severity    := Severity.DEBUG,
                        MessageCode := 0,
                        MessageText := 'Response.InvocationCounter = {1}',
                        Para1       :=  USINT_TO_STRING(_response.InvocationCounter));

// Create log entry for Reserve
CreateLogMessagePara1 ( Timestamp   := Timestamp,
                        MessageType := MessageType.CMD,
                        Severity    := Severity.DEBUG,
                        MessageCode := 0,
                        MessageText := 'Response.Reserve = {1}',
                        Para1       :=  SINT_TO_STRING(_response.Reserve));

// Create log entry for OriginID
CreateLogMessagePara1 ( Timestamp   := Timestamp,
                        MessageType := MessageType.CMD,
                        Severity    := Severity.DEBUG,
                        MessageCode := 0,
                        MessageText := 'Response.OriginID = {1}',
                        Para1       :=  INT_TO_STRING(_response.OriginID));
END_METHOD

METHOD PROTECTED Reset : DINT
VAR_INPUT
END_VAR
Reset := SUPER^.Reset();

Done               := FALSE;
Busy               := FALSE;
CommandBuffered    := FALSE;
CommandAborted     := FALSE;
CommandInterrupted := FALSE;
END_METHOD

END_FUNCTION_BLOCK

// Library/POUs/Additional/MC_UnitMeasurement/MC_UnitMeasurementFB
/// Measure the length of objects in the cartesian space, execution time for specified section of a job or signal output time of a specified signal
FUNCTION_BLOCK MC_UnitMeasurementFB EXTENDS RobotLibraryBaseEnableFB
// ------------------------------------------------------------------------- 
//  SRCI Robot Library                                                
// ------------------------------------------------------------------------- 
//                                                                           
//  Object:      UnitMeasurementFB                                       
//  Author:      Thorsten Brach                                                
//  Date:        2024-06-01
//
//  Description:                                              
//   
//                                                                           
//  Copyright: 
//    (C) 2024 Thorsten Brach. All rights reserved                                                                                                                                            
//             Licensed under the LGPL-3.0 license.
//                                                                           
//  Disclaimer:                                                                           
//    This project is provided without any guarantee and can be used for   
//    private and commercial purposes. Any use is at the user’s 
//    own risk and responsibility.
//
// -------------------------------------------------------------------------
VAR_INPUT
  /// command results
  ParCmd            : UnitMeasurementParCmd;
END_VAR

VAR_OUTPUT
  /// Command is transferred and confirmed by the RC
  CommandBuffered   : BOOL;
  /// Receiving of input parameter values has been acknowledged by RC
  ParameterAccepted : BOOL;
  /// command results
  OutCmd            : UnitMeasurementOutCmd;
END_VAR

VAR
  /// internal copy of command parameter 
 _parCmd            : UnitMeasurementParCmd;
  /// command data to send
 _command           : UnitMeasurementSendData;
  /// response data received
 _response          : UnitMeasurementRecvData;
  /// measurement number
 _measurementNo     : USINT; 
END_VAR

SUPER^(AxesGroup := AxesGroup);

METHOD PROTECTED CheckFunctionSupported : BOOL
VAR_IN_OUT
  /// Robot assignment of function
  AxesGroup : AxesGroup; 
END_VAR
CheckFunctionSupported := AxesGroup.InternalData.RCSupportedFunctions.UnitMeasurement;

IF ( NOT CheckFunctionSupported )
THEN
  // call base implementation for set error and create log entry
  SUPER^.CheckFunctionSupported(AxesGroup := AxesGroup);
END_IF
END_METHOD

METHOD PROTECTED CheckParameterChanged : BOOL
VAR_IN_OUT
  /// Robot assignment of function
  AxesGroup    : AxesGroup; 
END_VAR
// Check ParCmd Size is > 0, because MemCmp does not work correctly with size = 0
IF (SIZEOF(ParCmd) = 0) 
THEN 
  RETURN;
END_IF

// compare memory 
_parameterChanged := ( SysDepMemCmp(pData1 := ADR(ParCmd), pData2 := ADR(_parCmd), DataLen := SIZEOF(ParCmd)) <> RobotLibraryConstants.OK );

// check parameter valid ?
_parameterValid   := CheckParameterValid( AxesGroup := AxesGroup );

IF ((  _parameterChanged        )  AND 
    (  _parameterValid          )) OR
    (  _parameterUpdateInternal )  
THEN  
  // reset internal flag for send parameter update
 _parameterUpdateInternal := FALSE;
  // update internal copy of parameters 
 _parCmd := ParCmd;
  // inc parameter sequence
 _command.ParSeq := _command.ParSeq + 1;
  // update command data  
  CommandData := CreateCommandPayload(AxesGroup := AxesGroup); // ( Access via reference to rCommandFB in ACR )
  // notify active command register 
  AxesGroup.Acyclic.ActiveCommandRegister.NotifyParameterChanged := _uniqueID;
  // Reset parameter accepted flag
  ParameterAccepted := FALSE;  
END_IF
END_METHOD

METHOD INTERNAL CreateCommandPayload : RobotLibrarySendDataFB
VAR_IN_OUT
  /// Robot assignment of function
  AxesGroup : AxesGroup; 
END_VAR
// Table 6-803: Sent CMD payload (PLC to RC) of "UnitMeasurement"
// --------------------------
// Header
// --------------------------
// Byte 00 : UINT  - Type HB     
// Byte 01 :       - Type LB    
// Byte 02 : USINT - Reserve | ExecutionMode
// Byte 03 : USINT - ParSeq  | Priority
// --------------------------
// Datablock
// --------------------------
// Byte 04 : SINT   - EmitterID[0]
// Byte 05 : SINT   - EmitterID[1]
// Byte 06 : SINT   - EmitterID[2]
// Byte 07 : SINT   - EmitterID[3]
// Byte 08 : SINT   - ListenerID
// Byte 09 : BYTE   - Reserved
// Byte 10 : USINT  - TriggerMode
// Byte 11 : USINT  - MeasurementNo
// Byte 12 : USINT  - MeasuringMode
// set command parameter 
_command.CmdTyp          :=  CmdType.UnitMeasurement;
_command.ExecMode        :=  ExecMode;
_command.ParSeq          := _command.ParSeq;
_command.Priority        :=  Priority;
_command.EmitterID[0]    :=  0; {warning 'ToDo'}
_command.EmitterID[1]    :=  0; {warning 'ToDo'}
_command.EmitterID[2]    :=  0; {warning 'ToDo'}
_command.EmitterID[3]    :=  0; {warning 'ToDo'}
_command.ListenerID      :=  _parCmd.ListenerID;
_command.Reserve         :=  0;
_command.TriggerMode     :=  _parCmd.TriggerMode;
_command.MeasurementNo   :=  _measurementNo;
_command.MeasuringMode   :=  _parCmd.MeasuringMode;




// copy command data to header
_cmdHeader := _command;
// call base implementation to copy header to payload buffer
CreateCommandPayload := SUPER^.CreateCommandPayload(AxesGroup := AxesGroup);

// add command.EmitterID[0]
CreateCommandPayload.AddSint(_command.EmitterID[0]);
// add command.EmitterID[1]
CreateCommandPayload.AddSint(_command.EmitterID[1]);
// add command.EmitterID[2]
CreateCommandPayload.AddSint(_command.EmitterID[2]);
// add command.EmitterID[3]
CreateCommandPayload.AddSint(_command.EmitterID[3]);
// add command.ListenerID
CreateCommandPayload.AddSint(_command.ListenerID);
// add command.Reserved
CreateCommandPayload.AddByte(_command.Reserve);
// add command.TriggerMode
CreateCommandPayload.AddUsint(_command.TriggerMode);
// add command.MeasurementNo
CreateCommandPayload.AddUsint(_command.MeasurementNo);
// add command.MeasuringMode
CreateCommandPayload.AddUsint(_command.MeasuringMode);

// Create logging
CreateCommandPayloadLog(AxesGroup := AxesGroup);
END_METHOD

METHOD INTERNAL CreateCommandPayloadLog
VAR_IN_OUT
  /// Robot assignment of function
  AxesGroup : AxesGroup; 
END_VAR
VAR 
  /// internal index for loops
 _idx : DINT;
END_VAR
// Create log entry for Parameter start
CreateLogMessage      ( Timestamp   := AxesGroup.InternalData.SystemTime,
                        MessageType := MessageType.CMD,
                        Severity    := Severity.DEBUG,
                        MessageCode := 0,
                        MessageText := 'Create command payload with the following parameter(s) :');
  
// Create log entry for EmitterID[x]
FOR _idx := 0 TO 3
DO
  CreateLogMessagePara2 ( Timestamp   := AxesGroup.InternalData.SystemTime,
                          MessageType := MessageType.CMD,
                          Severity    := Severity.DEBUG,
                          MessageCode := 0,
                          MessageText := 'Command.EmitterID[{2}] = {1}',
                          Para1       :=  SINT_TO_STRING(_command.EmitterID[_idx]),
                          Para2       :=  DINT_TO_STRING(_idx));
END_FOR

// Create log entry for ListenerID
CreateLogMessagePara1 ( Timestamp   := AxesGroup.InternalData.SystemTime,
                        MessageType := MessageType.CMD,
                        Severity    := Severity.DEBUG,
                        MessageCode := 0,
                        MessageText := 'Command.ListenerID = {1}',
                        Para1       :=  SINT_TO_STRING(_command.ListenerID));
                        
// Create log entry for Reserve
CreateLogMessagePara1 ( Timestamp   := AxesGroup.InternalData.SystemTime,
                        MessageType := MessageType.CMD,
                        Severity    := Severity.DEBUG,
                        MessageCode := 0,
                        MessageText := 'Command.Reserve = {1}',
                        Para1       :=  BYTE_TO_STRING(_command.Reserve));
                        
// Create log entry for TriggerMode
CreateLogMessagePara1 ( Timestamp   := AxesGroup.InternalData.SystemTime,
                        MessageType := MessageType.CMD,
                        Severity    := Severity.DEBUG,
                        MessageCode := 0,
                        MessageText := 'Command.TriggerMode = {1}',
                        Para1       :=  TRIGGER_MODE_MEASUREMENT_TO_STRING(_command.TriggerMode));

// Create log entry for MeasurementNo
CreateLogMessagePara1 ( Timestamp   := AxesGroup.InternalData.SystemTime,
                        MessageType := MessageType.CMD,
                        Severity    := Severity.DEBUG,
                        MessageCode := 0,
                        MessageText := 'Command.MeasurementNo = {1}',
                        Para1       :=  USINT_TO_STRING(_command.MeasurementNo));

// Create log entry for MeasuringMode
CreateLogMessagePara1 ( Timestamp   := AxesGroup.InternalData.SystemTime,
                        MessageType := MessageType.CMD,
                        Severity    := Severity.DEBUG,
                        MessageCode := 0,
                        MessageText := 'Command.MeasuringMode = {1}',
                        Para1       :=  MEASUREING_UNIT_MODE_TO_STRING(_command.MeasuringMode));
END_METHOD

METHOD FB_init : BOOL
VAR_INPUT
  /// if TRUE, the retain variables are initialized (warm start / cold start)
  bInitRetains : BOOL; 
  /// if TRUE, the instance afterwards gets moved into the copy code (online change)
  bInCopyCode  : BOOL;  
END_VAR
MyType := 'MC_UnitMeasurementFB';

ExecMode := ExecutionMode.PARALLEL;
END_METHOD

METHOD PROTECTED OnCall
VAR_IN_OUT
  /// Robot assignment of function
  AxesGroup : AxesGroup; 
END_VAR
// call base implementation
SUPER^.OnCall(AxesGroup := AxesGroup);

CASE _stepCmd OF
  
  00:  IF ( _enable_R.Q )  
       THEN
         // reset the rising edge
        _enable_R();       
         // reset the falling edge
        _enable_F();      
         // Check function is supported and parameter are valid ?
         IF (( CheckFunctionSupported( AxesGroup := AxesGroup )) AND
             ( CheckParameterValid   ( AxesGroup := AxesGroup )))      
         THEN
           // set busy flag
           Busy := TRUE;
           // Reset command outputs
           SysDepMemSet(pDest := ADR(OutCmd), Value := 0, DataLen := SIZEOF(OutCmd));         
           // inc measurement number
          _measurementNo := _measurementNo + 1;
           // apply command parameter
          _parCmd := ParCmd;
           // init parameter sequence
          _command.ParSeq := 1;
           // create command data
           CommandData := CreateCommandPayload(AxesGroup := AxesGroup);
           // Add command to active command register
          _uniqueID := AxesGroup.Acyclic.ActiveCommandRegister.AddCmd( pCommandFB := ADR(THIS^ ));     
           // set timeout
           SetTimeout(PT := _timeoutCmd, rTimer := _timerCmd);
           // inc step counter
          _stepCmd := _stepCmd + 1;
         END_IF 
       END_IF
     

  01:  // Wait for responce received
       IF ( _responseReceived )
       THEN
         // reset response received flag
        _responseReceived := FALSE;

         CASE  _response.State 
         OF
           CmdMessageState.BUFFERED    : CommandBuffered    := TRUE;
           CmdMessageState.ACTIVE      : ParameterAccepted  := TRUE; 
                                         Enabled            := TRUE;          
           CmdMessageState.ERROR       : Error              := TRUE;
         END_CASE

         // Update results
         OutCmd.MeasurementActive := _response.MeasurementActive;
         OutCmd.Result            := _response.Result;
         OutCmd.OriginID          := _response.OriginID;
         OutCmd.InvocationCounter := _response.InvocationCounter;
                
         // Done, Aborted or Error ?
         IF (_response.State >= CmdMessageState.DONE )
         THEN
           // Reset Enabled flag
           Enabled := FALSE;
           // set timeout
           SetTimeout(PT := _timeoutCmd, rTimer := _timerCmd);
           // inc step counter
          _stepCmd := _stepCmd + 1; 
         END_IF
       END_IF

       // do not abort directly, so that the ParSeq update can be send
       IF ( _enable_R.Q ) OR ( _enable_F.Q ) 
       THEN
         // trigger parameter update to disable FB
        _parameterUpdateInternal := TRUE;
         // reset the rising edge
        _enable_R();       
         // reset the falling edge
        _enable_F();       
       END_IF

  02: IF (NOT Enable)
      THEN
        Reset();   
      END_IF

ELSE
  // invalid step
  ErrorID := RobotLibraryEvents.ERR_INVALID_STEP;
END_CASE


// Reset FB
IF (( _enable_R.Q ) OR
    ( _enable_F.Q ))
THEN
  Reset();
END_IF
END_METHOD

METHOD INTERNAL ParseResponsePayload : DINT
VAR_INPUT
  /// Response data
  ResponseData : RobotLibraryRecvDataFB;
  /// Timestamp
  Timestamp    : SystemTime;  
END_VAR
// Table 6-804: Received CMD payload (RC to PLC) of "UnitMeasurement"
// --------------------------
// Header
// --------------------------
// Byte 00 : USINT - ParSeq | State     
// Byte 01 : SINT  - AlarmMessageSeverity    
// Byte 02 : UINT  - AlarmMessageCode HB
// Byte 03 :       - AlarmMessageCode LB
// --------------------------
// Datablock
// --------------------------
// Byte 04 : USINT  - InvocationCounter
// Byte 05 : SINT   - Reserved
// Byte 06 : INT    - OriginID HW HB
// Byte 07 :        - OriginID HW LB
// Byte 08 : REAL   - Result HW HB
// Byte 09 :        - Result HW LB
// Byte 10 :        - Result LW HB
// Byte 11 :        - Result LW LB
// Byte 12 : BOOL   - MeasurementActive
// Byte 13 : USINT  - ResultNo
// --------------------------
// call base implementation to parse the header from payload buffer
ResponseData.PayloadPtr := SUPER^.ParseResponsePayload(ResponseData := ResponseData, Timestamp := Timestamp);

// copy parsed header to response
_response.ParSeq               := _rspHeader.ParSeq;
_response.State                := _rspHeader.State;
_response.AlarmMessageSeverity := _rspHeader.AlarmMessageSeverity;
_response.AlarmMessageCode     := _rspHeader.AlarmMessageCode;

// Get Response.InvocationCounter
_response.InvocationCounter := ResponseData.GetUsint();
// Get Response.Reserve
_response.Reserve := ResponseData.GetSint();
// Get Response.OriginID
_response.OriginID := ResponseData.GetInt();
// Get Response.Result
_response.Result := ResponseData.GetReal();
// Get Response.MeasurementActive
_response.MeasurementActive := ResponseData.GetBool();
// Get Response.ResultNo
_response.ResultNo := ResponseData.GetUsint();

// Create logging
ParseResponsePayloadLog(ResponseData := ResponseData, Timestamp := Timestamp);
END_METHOD

METHOD INTERNAL ParseResponsePayloadLog
VAR_INPUT
  /// Response data
  ResponseData : RobotLibraryRecvDataFB;
  /// Timestamp
  Timestamp    : SystemTime;  
END_VAR
// Create log entry for Parameter start
CreateLogMessage      ( Timestamp   := Timestamp,
                        MessageType := MessageType.CMD,
                        Severity    := Severity.DEBUG,
                        MessageCode := 0,
                        MessageText := 'Parsed the following parameter(s) from response data:');
                        
// Create log entry for InvocationCounter
CreateLogMessagePara1 ( Timestamp   := Timestamp,
                        MessageType := MessageType.CMD,
                        Severity    := Severity.DEBUG,
                        MessageCode := 0,
                        MessageText := 'Response.InvocationCounter = {1}',
                        Para1       :=  USINT_TO_STRING(_response.InvocationCounter));

// Create log entry for Reserve
CreateLogMessagePara1 ( Timestamp   := Timestamp,
                        MessageType := MessageType.CMD,
                        Severity    := Severity.DEBUG,
                        MessageCode := 0,
                        MessageText := 'Response.Reserve = {1}',
                        Para1       :=  SINT_TO_STRING(_response.Reserve));

// Create log entry for OriginID
CreateLogMessagePara1 ( Timestamp   := Timestamp,
                        MessageType := MessageType.CMD,
                        Severity    := Severity.DEBUG,
                        MessageCode := 0,
                        MessageText := 'Response.OriginID = {1}',
                        Para1       :=  INT_TO_STRING(_response.OriginID));

// Create log entry for Result
CreateLogMessagePara1 ( Timestamp   := Timestamp,
                        MessageType := MessageType.CMD,
                        Severity    := Severity.DEBUG,
                        MessageCode := 0,
                        MessageText := 'Response.Result = {1}',
                        Para1       :=  REAL_TO_STRING(_response.Result));

// Create log entry for MeasurementActive
CreateLogMessagePara1 ( Timestamp   := Timestamp,
                        MessageType := MessageType.CMD,
                        Severity    := Severity.DEBUG,
                        MessageCode := 0,
                        MessageText := 'Response.MeasurementActive = {1}',
                        Para1       :=  BOOL_TO_STRING(_response.MeasurementActive));

// Create log entry for ResultNo
CreateLogMessagePara1 ( Timestamp   := Timestamp,
                        MessageType := MessageType.CMD,
                        Severity    := Severity.DEBUG,
                        MessageCode := 0,
                        MessageText := 'Response.ResultNo = {1}',
                        Para1       :=  USINT_TO_STRING(_response.ResultNo));
END_METHOD

METHOD PROTECTED Reset : DINT
VAR_INPUT
END_VAR
Reset := SUPER^.Reset();

Busy               := FALSE;
CommandBuffered    := FALSE;
ParameterAccepted  := FALSE;
END_METHOD

END_FUNCTION_BLOCK

// Library/POUs/Additional/MC_WriteCallSubprogramCyclic/MC_WriteCallSubprogramCyclicFB
/// Writes cyclic data of called subprogram
FUNCTION_BLOCK MC_WriteCallSubprogramCyclicFB EXTENDS RobotLibraryBaseEnableFB
// ------------------------------------------------------------------------- 
//  SRCI Robot Library                                                
// ------------------------------------------------------------------------- 
//                                                                           
//  Object:      WriteCallSubprogramCyclicFB                                       
//  Author:      Thorsten Brach                                                
//  Date:        2024-06-01
//
//  Description:                                              
//   
//                                                                           
//  Copyright: 
//    (C) 2024 Thorsten Brach. All rights reserved                                                                                                                                            
//             Licensed under the LGPL-3.0 license.
//                                                                           
//  Disclaimer:                                                                           
//    This project is provided without any guarantee and can be used for   
//    private and commercial purposes. Any use is at the user’s 
//    own risk and responsibility.
//
// -------------------------------------------------------------------------
VAR_INPUT
  /// command parameter
  ParCmd  : WriteCallSubprogramCyclicParCmd;
END_VAR

VAR_OUTPUT
  /// command outputs
  OutCmd  : WriteCallSubprogramCyclicOutCmd;
END_VAR

SUPER^(AxesGroup := AxesGroup);

METHOD PROTECTED CheckFunctionSupported : BOOL
VAR_IN_OUT
  /// Robot assignment of function
  AxesGroup : AxesGroup; 
END_VAR
CheckFunctionSupported := AxesGroup.InternalData.RCSupportedFunctions.WriteCallSubprogramCyclic;

IF ( NOT CheckFunctionSupported )
THEN
  // call base implementation for set error and create log entry
  SUPER^.CheckFunctionSupported(AxesGroup := AxesGroup);
END_IF
END_METHOD

METHOD FB_init : BOOL
VAR_INPUT
  /// if TRUE, the retain variables are initialized (warm start / cold start)
  bInitRetains : BOOL; 
  /// if TRUE, the instance afterwards gets moved into the copy code (online change)
  bInCopyCode  : BOOL;  
END_VAR
MyType := 'MC_WriteCallSubprogramCyclicFB';
END_METHOD

METHOD PROTECTED OnCall
VAR_IN_OUT
  /// Robot assignment of function
  AxesGroup : AxesGroup; 
END_VAR
// call base implementation
SUPER^.OnCall(AxesGroup := AxesGroup);

AxesGroup.Parameter.Plc.OptionalCyclic.UseCallSubprogram := Enable;

Enabled := AxesGroup.CyclicOptional.PlcToRob.SubProgramData.Active;
Busy    := (Enabled <> Enable); 

AxesGroup.CyclicOptional.PlcToRob.SubProgramData.Data := ParCmd.Data;
END_METHOD

END_FUNCTION_BLOCK

// Library/POUs/AdvancedMove/MC_MoveApproachDirect/MC_MoveApproachDirectFB
/// Direct Move to target position through auxiliary position defined
/// by offset in all dimensions (movement to target posi tion PTP)
FUNCTION_BLOCK MC_MoveApproachDirectFB EXTENDS RobotLibraryBaseExecuteFB
// ------------------------------------------------------------------------- 
//  SRCI Robot Library                                                
// ------------------------------------------------------------------------- 
//                                                                           
//  Object:      MoveApproachDirectFB                                       
//  Author:      Thorsten Brach                                                
//  Date:        2024-06-01
//
//  Description:                                              
//   
//                                                                           
//  Copyright: 
//    (C) 2024 Thorsten Brach. All rights reserved                                                                                                                                            
//             Licensed under the LGPL-3.0 license.
//                                                                           
//  Disclaimer:                                                                           
//    This project is provided without any guarantee and can be used for   
//    private and commercial purposes. Any use is at the user’s 
//    own risk and responsibility.
//
// -------------------------------------------------------------------------
VAR_INPUT
  /// Parameter which determines the behavior towards the previously sent and still active or buffered commands
  AbortingMode       : AbortingMode;
  /// Defines the target sequence in which the command will be executed
  SequenceFlag       : SequenceFlag;
  /// command parameter
  ParCmd             : MoveApproachDirectParCmd;       
END_VAR

VAR_OUTPUT
  /// Command is transferred and confirmed by the RC
  CommandBuffered    : BOOL;
  /// The command takes control of the motion of the according axis group
  Active             : BOOL;
  /// The command was aborted by another command.
  CommandAborted     : BOOL;
  /// TRUE, while command is interrupted during execution and can be continued
  CommandInterrupted : BOOL;
  /// command results
  OutCmd             : MoveApproachDirectOutCmd;     
END_VAR

VAR
  /// internal copy of command parameter 
 _parCmd             : MoveApproachDirectParCmd;
  /// command data to send
 _command            : MoveApproachDirectSendData;
  /// response data received
 _response           : MoveApproachDirectRecvData;      
END_VAR

SUPER^(AxesGroup := AxesGroup);

METHOD PROTECTED CheckFunctionSupported : BOOL
VAR_IN_OUT
  /// Robot assignment of function
  AxesGroup : AxesGroup; 
END_VAR
CheckFunctionSupported := AxesGroup.InternalData.RCSupportedFunctions.MoveApproachDirect;

IF ( NOT CheckFunctionSupported )
THEN
  // call base implementation for set error and create log entry
  SUPER^.CheckFunctionSupported(AxesGroup := AxesGroup);
END_IF
END_METHOD

METHOD PROTECTED CheckParameterChanged : BOOL
VAR_IN_OUT
  /// Robot assignment of function
  AxesGroup    : AxesGroup; 
END_VAR
// Check ParCmd Size is > 0, because MemCmp does not work correctly with size = 0
IF (SIZEOF(ParCmd) = 0) 
THEN 
  RETURN;
END_IF

// compare memory 
_parameterChanged := ( SysDepMemCmp(pData1 := ADR(ParCmd), pData2 := ADR(_parCmd), DataLen := SIZEOF(ParCmd)) <> RobotLibraryConstants.OK );

// check parameter valid ?
_parameterValid   := CheckParameterValid( AxesGroup := AxesGroup );

IF ((  _parameterChanged        )  AND 
    (  _parameterValid          )) OR
    (  _parameterUpdateInternal )  
THEN  
  // reset internal flag for send parameter update
 _parameterUpdateInternal := FALSE;
  // update internal copy of parameters 
 _parCmd := ParCmd;
  // inc parameter sequence
 _command.ParSeq := _command.ParSeq + 1;
  // update command data  
  CommandData := CreateCommandPayload(AxesGroup := AxesGroup); // ( Access via reference to rCommandFB in ACR )
  // notify active command register 
  AxesGroup.Acyclic.ActiveCommandRegister.NotifyParameterChanged := _uniqueID;
END_IF
END_METHOD

METHOD INTERNAL CreateCommandPayload : RobotLibrarySendDataFB
VAR_IN_OUT
  /// Robot assignment of function
  AxesGroup : AxesGroup; 
END_VAR
// Table 6-387: Sent CMD payload (PLC to RC) of "MoveApproachDirect"
// --------------------------
// Header
// --------------------------
// Byte 00 : UINT  - Type HB     
// Byte 01 :       - Type LB    
// Byte 02 : USINT - Reserve | ExecutionMode
// Byte 03 : USINT - ParSeq  | Priority
// --------------------------
// Datablock
// --------------------------
// Byte 04 : SINT      - EmitterID[0]
// Byte 05 : SINT      - EmitterID[1]
// Byte 06 : SINT      - EmitterID[2]
// Byte 07 : SINT      - EmitterID[3]
// Byte 08 : SINT      - ListenerID
// Byte 09 : BYTE      - Reserved
// Byte 10 : UINT      - VelocityRate LW HB
// Byte 11 :           - VelocityRate LW LB
// Byte 12 : UINT      - AccelerationRate LW HB
// Byte 13 :           - AccelerationRate LW LB
// Byte 14 : UINT      - DecelerationRate LW HB
// Byte 15 :           - DecelerationRate LW LB
// Byte 16 : UINT      - JerkRate LW HB
// Byte 17 :           - JerkRate LW LB
// Byte 18 : USINT     - ToolNo
// Byte 19 : USINT     - FrameNo
// Byte 20 : USINT     - BlendingMode
// Byte 21 : USINT     - OriMode
// Byte 22 : REAL      - BlendingParameter[0] HW HB
// Byte 23 :           - BlendingParameter[0] HW LB
// Byte 24 :           - BlendingParameter[0] LW HB
// Byte 25 :           - BlendingParameter[0] LW LB
// Byte 26 : REAL      - BlendingParameter[1] HW HB
// Byte 27 :           - BlendingParameter[1] HW LB
// Byte 28 :           - BlendingParameter[1] LW HB
// Byte 29 :           - BlendingParameter[1] LW LB
// Byte 30 : REAL      - TargetPosition.X HW HB
// Byte 31 :           - TargetPosition.X HW LB
// Byte 32 :           - TargetPosition.X LW HB
// Byte 33 :           - TargetPosition.X LW LB
// Byte 34 : REAL      - TargetPosition.Y HW HB
// Byte 35 :           - TargetPosition.Y HW LB
// Byte 36 :           - TargetPosition.Y LW HB
// Byte 37 :           - TargetPosition.Y LW LB
// Byte 38 : REAL      - TargetPosition.Z HW HB
// Byte 39 :           - TargetPosition.Z HW LB
// Byte 40 :           - TargetPosition.Z LW HB
// Byte 41 :           - TargetPosition.Z LW LB
// Byte 42 : REAL      - TargetPosition.RX HW HB
// Byte 43 :           - TargetPosition.RX HW LB
// Byte 44 :           - TargetPosition.RX LW HB
// Byte 45 :           - TargetPosition.RX LW LB
// Byte 46 : REAL      - TargetPosition.RY HW HB
// Byte 47 :           - TargetPosition.RY HW LB
// Byte 48 :           - TargetPosition.RY LW HB
// Byte 49 :           - TargetPosition.RY LW LB
// Byte 50 : REAL      - TargetPosition.RZ HW HB
// Byte 51 :           - TargetPosition.RZ HW LB
// Byte 52 :           - TargetPosition.RZ LW HB
// Byte 53 :           - TargetPosition.RZ LW LB
// Byte 54 : ArmConfig - Config
// Byte 55 :           - Reserved
// Byte 56 : BYTE      - TargetPosition.TurnNumber[0]
// Byte 57 : BYTE      - TargetPosition.TurnNumber[1]
// Byte 58 : BYTE      - TargetPosition.TurnNumber[2]
// Byte 59 : BYTE      - TargetPosition.TurnNumber[3]
// Byte 60 : REAL      - TargetPosition.E1 HW HB
// Byte 61 :           - TargetPosition.E1 HW LB
// Byte 62 :           - TargetPosition.E1 LW HB
// Byte 63 :           - TargetPosition.E1 LW LB
// Byte 64 : REAL      - Offset.X HW HB
// Byte 65 :           - Offset.X HW LB
// Byte 66 :           - Offset.X LW HB
// Byte 67 :           - Offset.X LW LB
// Byte 68 : REAL      - Offset.Y HW HB
// Byte 69 :           - Offset.Y HW LB
// Byte 70 :           - Offset.Y LW HB
// Byte 71 :           - Offset.Y LW LB
// Byte 72 : REAL      - Offset.Z HW HB
// Byte 73 :           - Offset.Z HW LB
// Byte 74 :           - Offset.Z LW HB
// Byte 75 :           - Offset.Z LW LB
// Byte 76 : REAL      - Offset.RX HW HB
// Byte 77 :           - Offset.RX HW LB
// Byte 78 :           - Offset.RX LW HB
// Byte 79 :           - Offset.RX LW LB
// Byte 80 : REAL      - Offset.RY HW HB
// Byte 81 :           - Offset.RY HW LB
// Byte 82 :           - Offset.RY LW HB
// Byte 83 :           - Offset.RY LW LB
// Byte 84 : REAL      - Offset.RZ HW HB
// Byte 85 :           - Offset.RZ HW LB
// Byte 86 :           - Offset.RZ LW HB
// Byte 87 :           - Offset.RZ LW LB
// Byte 88 : REAL      - AuxCornerDistance HW HB
// Byte 89 :           - AuxCornerDistance HW LB
// Byte 90 :           - AuxCornerDistance LW HB
// Byte 91 :           - AuxCornerDistance LW LB
// Byte 92 : REAL      - VelocityCoefficient HW HB
// Byte 93 :           - VelocityCoefficient HW LB
// Byte 94 :           - VelocityCoefficient LW HB
// Byte 95 :           - VelocityCoefficient LW LB
// Byte 96 : BOOL      - Manipulation
// Byte 97 : BYTE      - ConfigMode[0]
// Byte 98 : BYTE      - ConfigMode[1]
// Byte 99 : USINT     - TurnMode
// Byte 100: USINT     - ReferenceType
// Byte 101: UINT      - Time LW HB
// Byte 102:           - Time LW LB
// Byte 103: REAL      - TargetPosition.E2 HW HB
// Byte 104:           - TargetPosition.E2 HW LB
// Byte 105:           - TargetPosition.E2 LW HB
// Byte 106:           - TargetPosition.E2 LW LB
// Byte 107: REAL      - TargetPosition.E3 HW HB
// Byte 108:           - TargetPosition.E3 HW LB
// Byte 109:           - TargetPosition.E3 LW HB
// Byte 110:           - TargetPosition.E3 LW LB
// Byte 111: REAL      - TargetPosition.E4 HW HB
// Byte 112:           - TargetPosition.E4 HW LB
// Byte 113:           - TargetPosition.E4 LW HB
// Byte 114:           - TargetPosition.E4 LW LB
// Byte 115: REAL      - TargetPosition.E5 HW HB
// Byte 116:           - TargetPosition.E5 HW LB
// Byte 117:           - TargetPosition.E5 LW HB
// Byte 118:           - TargetPosition.E5 LW LB
// Byte 119: REAL      - TargetPosition.E6 HW HB
// Byte 120:           - TargetPosition.E6 HW LB
// Byte 121:           - TargetPosition.E6 LW HB
// Byte 122:           - TargetPosition.E6 LW LB
// set command parameter 
_command.CmdTyp                    :=  CmdType.MoveApproachDirect;
_command.ExecMode                  :=  ExecMode;
_command.ParSeq                    := _command.ParSeq;
_command.Priority                  :=  Priority;
_command.EmitterID[0]              := _parCmd.EmitterID[0];
_command.EmitterID[1]              := _parCmd.EmitterID[1];
_command.EmitterID[2]              := _parCmd.EmitterID[2];
_command.EmitterID[3]              := _parCmd.EmitterID[3];
_command.ListenerID                := 0; {warning 'ToDo'}
_command.Reserve                   := 0;
_command.VelocityRate              := REAL_TO_PERCENT_UINT(_parCmd.VelocityRate     , IsOptional := FALSE);
_command.AccelerationRate          := REAL_TO_PERCENT_UINT(_parCmd.AccelerationRate , IsOptional := FALSE);
_command.DecelerationRate          := REAL_TO_PERCENT_UINT(_parCmd.DecelerationRate , IsOptional := TRUE );
_command.JerkRate                  := REAL_TO_PERCENT_UINT(_parCmd.JerkRate         , IsOptional := TRUE );
_command.ToolNo                    := _parCmd.ToolNo;
_command.FrameNo                   := _parCmd.FrameNo;
_command.BlendingMode              := _parCmd.BlendingMode;
_command.OriMode                   := _parCmd.OriMode;
_command.BlendingParameter         := _parCmd.BlendingParameter;
_command.TargetPosition            := _parCmd.TargetPosition;
_command.Offset                    := _parCmd.Offset;
_command.AuxCornerDistance         := _parCmd.AuxCornerDistance;
_command.VelocityCoefficient       := _parCmd.VelocityCoefficient;
_command.Manipulation              := _parCmd.Manipulation;
_command.ConfigMode                :=  ArmConfigParameterToBytes(_parCmd.ConfigMode);
_command.TurnMode                  := _parCmd.TurnMode;
_command.ReferenceType             := _parCmd.ReferenceType;
_command.MoveTime                  := TIME_TO_UINT(_parCmd.MoveTime);


// copy command data to header
_cmdHeader := _command;
// call base implementation to copy header to payload buffer
CreateCommandPayload := SUPER^.CreateCommandPayload(AxesGroup := AxesGroup);

// add command.EmitterID[0]
CreateCommandPayload.AddSint(_command.EmitterID[0]);
// add command.EmitterID[1]
CreateCommandPayload.AddSint(_command.EmitterID[1]);
// add command.EmitterID[2]
CreateCommandPayload.AddSint(_command.EmitterID[2]);
// add command.EmitterID[3]
CreateCommandPayload.AddSint(_command.EmitterID[3]);
// add command.ListenerID
CreateCommandPayload.AddSint(_command.ListenerID);
// add command.Reserve
CreateCommandPayload.AddByte(_command.Reserve);
// add command.VelocityRate
CreateCommandPayload.AddUint(_command.VelocityRate);
// add command.AccelerationRate
CreateCommandPayload.AddUint(_command.AccelerationRate);
// add command.DecelerationRate
CreateCommandPayload.AddUint(_command.DecelerationRate);
// add command.JerkRate
CreateCommandPayload.AddUint(_command.JerkRate);
// add command.ToolNo
CreateCommandPayload.AddUsint(_command.ToolNo);
// add command.FrameNo
CreateCommandPayload.AddUsint(_command.FrameNo);
// add command.BlendingMode
CreateCommandPayload.AddUsint(_command.BlendingMode);
// add command.OriMode
CreateCommandPayload.AddUsint(_command.OriMode);
// add command.BlendingParameter[0]
CreateCommandPayload.AddReal(_command.BlendingParameter[0]);
// add command.BlendingParameter[1]
CreateCommandPayload.AddReal(_command.BlendingParameter[1]);
// add command.TargetPosition.X
CreateCommandPayload.AddReal(_command.TargetPosition.X);
// add command.TargetPosition.Y
CreateCommandPayload.AddReal(_command.TargetPosition.Y);
// add command.TargetPosition.Z
CreateCommandPayload.AddReal(_command.TargetPosition.Z);
// add command.TargetPosition.Rx
CreateCommandPayload.AddReal(_command.TargetPosition.Rx);
// add command.TargetPosition.Ry
CreateCommandPayload.AddReal(_command.TargetPosition.Ry);
// add command.TargetPosition.Rz
CreateCommandPayload.AddReal(_command.TargetPosition.Rz);
// add command.TargetPosition.Config
CreateCommandPayload.AddArmConfig(_command.TargetPosition.Config);
// add command.Reserve
CreateCommandPayload.AddByte(_command.Reserve);
// add command.TargetPosition.TurnNumber
CreateCommandPayload.AddTurnNumber(_command.TargetPosition.TurnNumber);
// add command.TargetPosition.E1
CreateCommandPayload.AddReal(_command.TargetPosition.E1);
// add command.Offset.X
CreateCommandPayload.AddReal(_command.Offset.X);
// add command.Offset.Y
CreateCommandPayload.AddReal(_command.Offset.Y);
// add command.Offset.Z
CreateCommandPayload.AddReal(_command.Offset.Z);
// add command.Offset.Rx
CreateCommandPayload.AddReal(_command.Offset.Rx);
// add command.Offset.Ry
CreateCommandPayload.AddReal(_command.Offset.Ry);
// add command.Offset.Rz
CreateCommandPayload.AddReal(_command.Offset.Rz); {warning 'ToDo'}
// add command.AuxCornerDistance
CreateCommandPayload.AddReal(_command.AuxCornerDistance);
// add command.VelocityCoefficient
CreateCommandPayload.AddReal(_command.VelocityCoefficient);
// add command.Manipulation
CreateCommandPayload.AddBool(_command.Manipulation);
// add command.ConfigMode[0]
CreateCommandPayload.AddByte(_command.ConfigMode[0]);
// add command.ConfigMode[1]
CreateCommandPayload.AddByte(_command.ConfigMode[1]);
// add command.TurnMode
CreateCommandPayload.AddUsint(_command.TurnMode);
// add command.ReferenceType
CreateCommandPayload.AddUsint(_command.ReferenceType);
// add command.MoveTime
CreateCommandPayload.AddUint(_command.MoveTime);
// add command.TargetPosition.E2
CreateCommandPayload.AddReal(_command.TargetPosition.E2);
// add command.TargetPosition.E3
CreateCommandPayload.AddReal(_command.TargetPosition.E3);
// add command.TargetPosition.E4
CreateCommandPayload.AddReal(_command.TargetPosition.E4);
// add command.TargetPosition.E5
CreateCommandPayload.AddReal(_command.TargetPosition.E5);
// add command.TargetPosition.E6
CreateCommandPayload.AddReal(_command.TargetPosition.E6);

// Create logging
CreateCommandPayloadLog(AxesGroup := AxesGroup);
END_METHOD

METHOD INTERNAL CreateCommandPayloadLog
VAR_IN_OUT
  /// Robot assignment of function
  AxesGroup : AxesGroup; 
END_VAR
VAR 
  /// internal index for loops
 _idx : DINT;
END_VAR
// Create log entry for Parameter start
CreateLogMessage      ( Timestamp   := AxesGroup.InternalData.SystemTime,
                        MessageType := MessageType.CMD,
                        Severity    := Severity.DEBUG,
                        MessageCode := 0,
                        MessageText := 'Create command payload with the following parameter(s) :');
  
// Create log entry for EmitterID[x]
FOR _idx := 0 TO 3
DO
  CreateLogMessagePara2 ( Timestamp   := AxesGroup.InternalData.SystemTime,
                          MessageType := MessageType.CMD,
                          Severity    := Severity.DEBUG,
                          MessageCode := 0,
                          MessageText := 'Command.EmitterID[{2}] = {1}',
                          Para1       :=  SINT_TO_STRING(_command.EmitterID[_idx]),
                          Para2       :=  DINT_TO_STRING(_idx));
END_FOR

// Create log entry for ListenerID
CreateLogMessagePara1 ( Timestamp   := AxesGroup.InternalData.SystemTime,
                        MessageType := MessageType.CMD,
                        Severity    := Severity.DEBUG,
                        MessageCode := 0,
                        MessageText := 'Command.ListenerID = {1}',
                        Para1       :=  SINT_TO_STRING(_command.ListenerID));
                        
// Create log entry for Reserve
CreateLogMessagePara1 ( Timestamp   := AxesGroup.InternalData.SystemTime,
                        MessageType := MessageType.CMD,
                        Severity    := Severity.DEBUG,
                        MessageCode := 0,
                        MessageText := 'Command.Reserve = {1}',
                        Para1       :=  BYTE_TO_STRING(_command.Reserve));

// Create log entry for VelocityRate
CreateLogMessagePara1 ( Timestamp   := AxesGroup.InternalData.SystemTime,
                        MessageType := MessageType.CMD,
                        Severity    := Severity.DEBUG,
                        MessageCode := 0,
                        MessageText := 'Command.VelocityRate = {1}',
                        Para1       :=  UINT_TO_STRING(_command.VelocityRate));

// Create log entry for AccelerationRate
CreateLogMessagePara1 ( Timestamp   := AxesGroup.InternalData.SystemTime,
                        MessageType := MessageType.CMD,
                        Severity    := Severity.DEBUG,
                        MessageCode := 0,
                        MessageText := 'Command.AccelerationRate = {1}',
                        Para1       :=  UINT_TO_STRING(_command.AccelerationRate));
                        
// Create log entry for DecelerationRate
CreateLogMessagePara1 ( Timestamp   := AxesGroup.InternalData.SystemTime,
                        MessageType := MessageType.CMD,
                        Severity    := Severity.DEBUG,
                        MessageCode := 0,
                        MessageText := 'Command.DecelerationRate = {1}',
                        Para1       :=  UINT_TO_STRING(_command.DecelerationRate));

// Create log entry for JerkRate
CreateLogMessagePara1 ( Timestamp   := AxesGroup.InternalData.SystemTime,
                        MessageType := MessageType.CMD,
                        Severity    := Severity.DEBUG,
                        MessageCode := 0,
                        MessageText := 'Command.JerkRate = {1}',
                        Para1       :=  UINT_TO_STRING(_command.JerkRate));

// Create log entry for ToolNo
CreateLogMessagePara1 ( Timestamp   := AxesGroup.InternalData.SystemTime,
                        MessageType := MessageType.CMD,
                        Severity    := Severity.DEBUG,
                        MessageCode := 0,
                        MessageText := 'Command.ToolNo = {1}',
                        Para1       :=  USINT_TO_STRING(_command.ToolNo));

// Create log entry for FrameNo
CreateLogMessagePara1 ( Timestamp   := AxesGroup.InternalData.SystemTime,
                        MessageType := MessageType.CMD,
                        Severity    := Severity.DEBUG,
                        MessageCode := 0,
                        MessageText := 'Command.FrameNo = {1}',
                        Para1       :=  USINT_TO_STRING(_command.FrameNo));

// Create log entry for BlendingMode
CreateLogMessagePara1 ( Timestamp   := AxesGroup.InternalData.SystemTime,
                        MessageType := MessageType.CMD,
                        Severity    := Severity.DEBUG,
                        MessageCode := 0,
                        MessageText := 'Command.BlendingMode = {1}',
                        Para1       :=  BLENDING_MODE_TO_STRING(_command.BlendingMode));

// Create log entry for OriMode
CreateLogMessagePara1 ( Timestamp   := AxesGroup.InternalData.SystemTime,
                        MessageType := MessageType.CMD,
                        Severity    := Severity.DEBUG,
                        MessageCode := 0,
                        MessageText := 'Command.OriMode = {1}',
                        Para1       :=  ORI_MODE_TO_STRING(_command.OriMode));

// Create log entry for BlendingParameter[0]
CreateLogMessagePara1 ( Timestamp   := AxesGroup.InternalData.SystemTime,
                        MessageType := MessageType.CMD,
                        Severity    := Severity.DEBUG,
                        MessageCode := 0,
                        MessageText := 'Command.BlendingParameter[0] = {1}',
                        Para1       :=  REAL_TO_STRING(_command.BlendingParameter[0]));

// Create log entry for BlendingParameter[1]
CreateLogMessagePara1 ( Timestamp   := AxesGroup.InternalData.SystemTime,
                        MessageType := MessageType.CMD,
                        Severity    := Severity.DEBUG,
                        MessageCode := 0,
                        MessageText := 'Command.BlendingParameter[1] = {1}',
                        Para1       :=  REAL_TO_STRING(_command.BlendingParameter[1]));

// Create log entry for TargetPosition.X
CreateLogMessagePara1 ( Timestamp   := AxesGroup.InternalData.SystemTime,
                        MessageType := MessageType.CMD,
                        Severity    := Severity.DEBUG,
                        MessageCode := 0,
                        MessageText := 'Command.TargetPosition.X = {1}',
                        Para1       :=  REAL_TO_STRING(_command.TargetPosition.X));

// Create log entry for TargetPosition.Y
CreateLogMessagePara1 ( Timestamp   := AxesGroup.InternalData.SystemTime,
                        MessageType := MessageType.CMD,
                        Severity    := Severity.DEBUG,
                        MessageCode := 0,
                        MessageText := 'Command.TargetPosition.Y = {1}',
                        Para1       :=  REAL_TO_STRING(_command.TargetPosition.Y));

